FUNCTION_BLOCK SERVER (* SERVER Function Block Type for Central Server ME Algorithm *)
  (* Standard: 61499-2 *)
  (* Version 0.2, 2003-12-04, JHC, Rockwell Automation, Renamed for better indexing. *)
  (* Version 0.1, 2002-11-05, JHC, Rockwell Automation, Corrected missing ST element in Algorithm REQ. *)
  (* Version 0.0, 2000-05-30, JHC, Rockwell Automation *)
  (* Compiler header: package fb.rt.cs725; *)
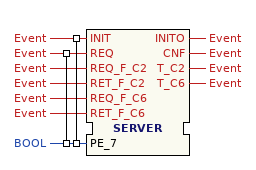
  EVENT_INPUT
    INIT WITH PE_7; (* Initialization Request *)
    REQ WITH PE_7; (* Normal Execution Request *)
    REQ_F_C2;
    RET_F_C2;
    REQ_F_C6;
    RET_F_C6;
  END_EVENT
  EVENT_OUTPUT
    INITO; (* Initialization Confirm *)
    CNF; (* Execution Confirmation *)
    T_C2;
    T_C6;
  END_EVENT
  VAR_INPUT
    PE_7 : BOOL; (* Input event qualifier *)
  END_VAR
  VAR
    C2_FLAG : BOOL;
    C6_FLAG : BOOL;
    PRIORITY : BOOL;
  END_VAR
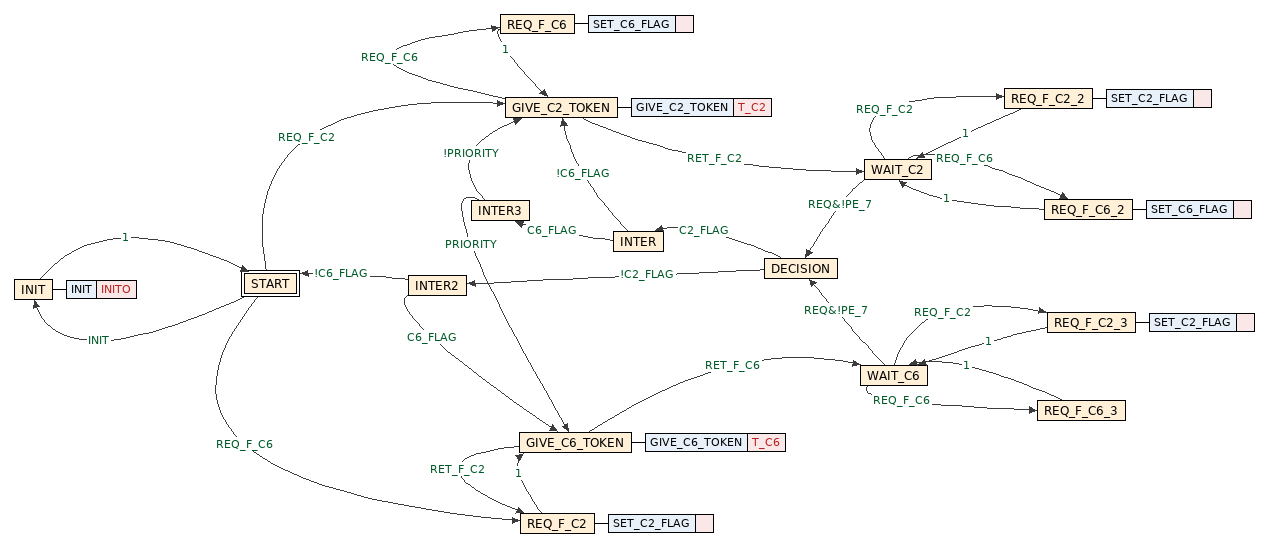
  EC_STATES
    START; (* Initial State *)
    INIT : INIT -> INITO; (* Initialization *)
    GIVE_C2_TOKEN : GIVE_C2_TOKEN -> T_C2;
    REQ_F_C6 : SET_C6_FLAG;
    WAIT_C2;
    DECISION;
    GIVE_C6_TOKEN : GIVE_C6_TOKEN -> T_C6;
    WAIT_C6;
    INTER;
    INTER2;
    INTER3;
    REQ_F_C2 : SET_C2_FLAG;
    REQ_F_C2_2 : SET_C2_FLAG;
    REQ_F_C6_2 : SET_C6_FLAG;
    REQ_F_C2_3 : SET_C2_FLAG;
    REQ_F_C6_3;
  END_STATES
  EC_TRANSITIONS
    START TO INIT := INIT;
    INIT TO START := 1;
    GIVE_C2_TOKEN TO REQ_F_C6 := REQ_F_C6;
    REQ_F_C6 TO GIVE_C2_TOKEN := 1;
    GIVE_C2_TOKEN TO WAIT_C2 := RET_F_C2;
    WAIT_C2 TO DECISION := REQ&!PE_7;
    GIVE_C6_TOKEN TO WAIT_C6 := RET_F_C6;
    WAIT_C6 TO DECISION := REQ&!PE_7;
    DECISION TO INTER := C2_FLAG;
    DECISION TO INTER2 := !C2_FLAG;
    INTER2 TO START := !C6_FLAG;
    INTER2 TO GIVE_C6_TOKEN := C6_FLAG;
    INTER TO GIVE_C2_TOKEN := !C6_FLAG;
    INTER TO INTER3 := C6_FLAG;
    INTER3 TO GIVE_C2_TOKEN := !PRIORITY;
    INTER3 TO GIVE_C6_TOKEN := PRIORITY;
    GIVE_C6_TOKEN TO REQ_F_C2 := RET_F_C2;
    REQ_F_C2 TO GIVE_C6_TOKEN := 1;
    WAIT_C2 TO REQ_F_C2_2 := REQ_F_C2;
    REQ_F_C2_2 TO WAIT_C2 := 1;
    WAIT_C2 TO REQ_F_C6_2 := REQ_F_C6;
    REQ_F_C6_2 TO WAIT_C2 := 1;
    WAIT_C6 TO REQ_F_C2_3 := REQ_F_C2;
    REQ_F_C2_3 TO WAIT_C6 := 1;
    REQ_F_C6_3 TO WAIT_C6 := 1;
    WAIT_C6 TO REQ_F_C6_3 := REQ_F_C6;
    START TO GIVE_C2_TOKEN := REQ_F_C2;
    START TO REQ_F_C2 := REQ_F_C6;
  END_TRANSITIONS
  ALGORITHM INIT IN ST: (* Initialization algorithm *)

  END_ALGORITHM
  ALGORITHM REQ IN ST: (* Normally executed algorithm *)

  END_ALGORITHM
  ALGORITHM GIVE_C2_TOKEN IN Java:
C2_FLAG.value = false;
System.out.println("-------------------");
System.out.println("GIVE TOKEN TO C2!!");
System.out.println("-------------------");
  END_ALGORITHM
  ALGORITHM SET_C6_FLAG IN Java:
C6_FLAG.value = true;
if(C2_FLAG.value){
PRIORITY.value = false;
} else {
PRIORITY.value = true;
}
  END_ALGORITHM
  ALGORITHM GIVE_C6_TOKEN IN Java:
C6_FLAG.value = false;
System.out.println("-------------------");
System.out.println("GIVE TOKEN TO C6!!");
System.out.println("-------------------");
  END_ALGORITHM
  ALGORITHM SET_C2_FLAG IN Java:
C2_FLAG.value = true;
if(C6_FLAG.value){
PRIORITY.value = true;
} else {
PRIORITY.value = false;
}
  END_ALGORITHM
END_FUNCTION_BLOCK
